FUNCTION_BLOCK DepotSkill (* Basic FB with empty ECC *)
  (* Standard: 61499-2 *)
  (* Version 1.0, 2021-09-15, dorofeev *)
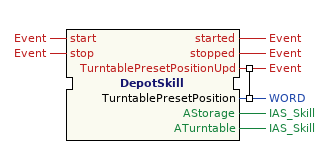
  EVENT_INPUT
    start;
    stop;
  END_EVENT
  EVENT_OUTPUT
    started;
    stopped;
    TurntablePresetPositionUpd WITH TurntablePresetPosition;
  END_EVENT
  VAR_OUTPUT
    TurntablePresetPosition : WORD;
  END_VAR
  PLUGS
    AStorage : IAS_Skill;
    ATurntable : IAS_Skill;
  END_PLUGS
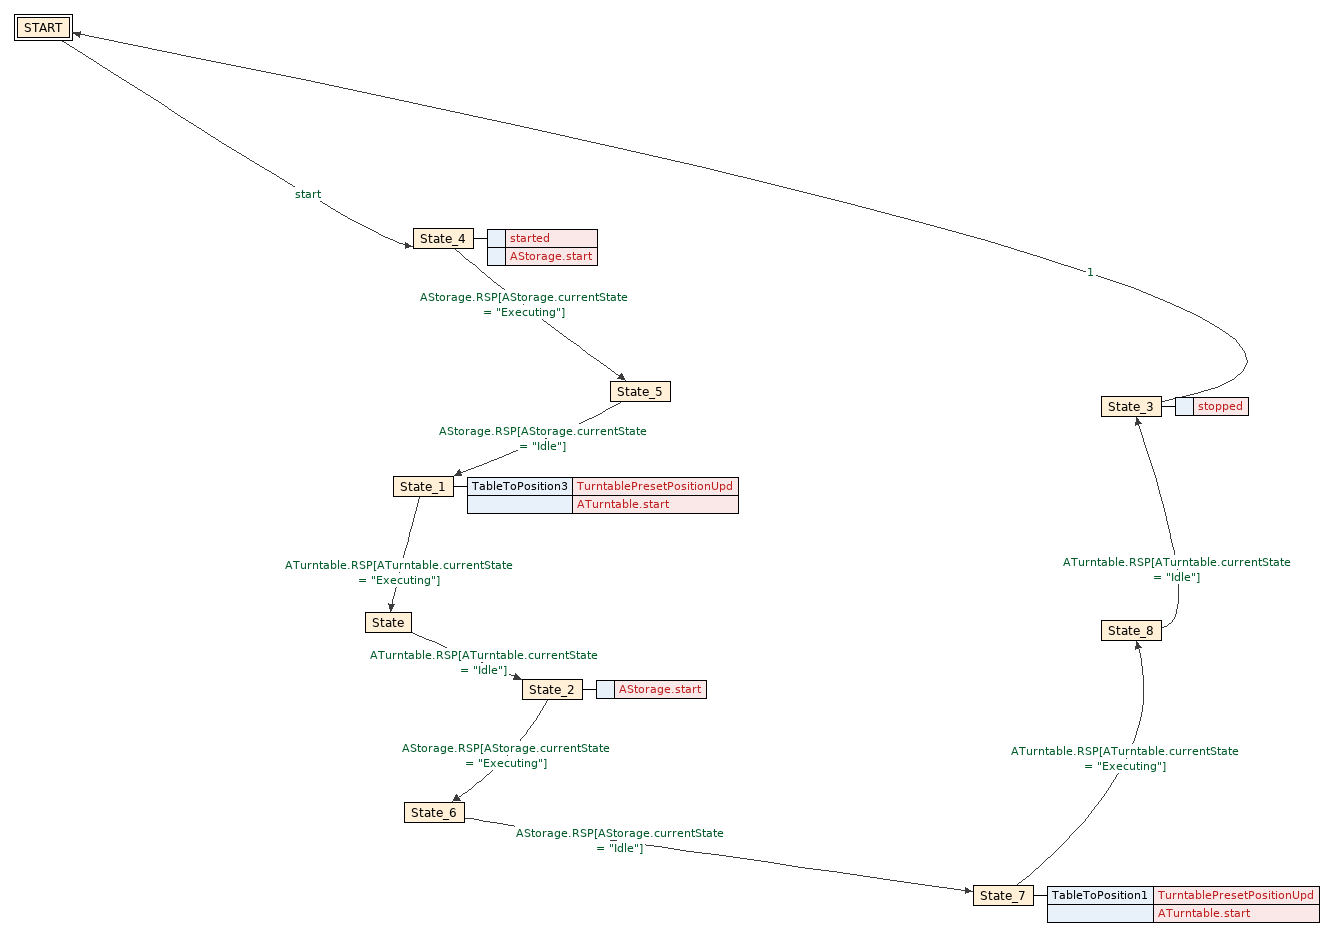
  EC_STATES
    START; (* Initial State *)
    State_1 : TableToPosition3 -> TurntablePresetPositionUpd, -> ATurntable.start;
    State_2 : -> AStorage.start;
    State_3 : -> stopped;
    State_4 : -> started, -> AStorage.start;
    State;
    State_5;
    State_6;
    State_7 : TableToPosition1 -> TurntablePresetPositionUpd, -> ATurntable.start;
    State_8;
  END_STATES
  EC_TRANSITIONS
    START TO State_4 := start;
    State_3 TO START := 1;
    State_1 TO State := ATurntable.RSP[ATurntable.currentState = "Executing"];
    State TO State_2 := ATurntable.RSP[ATurntable.currentState = "Idle"];
    State_4 TO State_5 := AStorage.RSP[AStorage.currentState = "Executing"];
    State_5 TO State_1 := AStorage.RSP[AStorage.currentState = "Idle"];
    State_2 TO State_6 := AStorage.RSP[AStorage.currentState = "Executing"];
    State_6 TO State_7 := AStorage.RSP[AStorage.currentState = "Idle"];
    State_7 TO State_8 := ATurntable.RSP[ATurntable.currentState = "Executing"];
    State_8 TO State_3 := ATurntable.RSP[ATurntable.currentState = "Idle"];
  END_TRANSITIONS
  ALGORITHM TableToPosition3 IN ST: (* New Algorithm *)
TurntablePresetPosition := 3;
  END_ALGORITHM
  ALGORITHM TableToPosition1 IN ST: (* New Algorithm *)
TurntablePresetPosition := 1;
  END_ALGORITHM
END_FUNCTION_BLOCK
